// TIA Portal V17 export
// export: Created 2024-08-07T21:43:56.755599Z, ExportSetting WithDefaults, DisplayName Totally Integrated Automation Portal, DisplayVersion V17 Update 7, DisplayName TIA Portal Openness, DisplayVersion V17 Update 7, DisplayName TIA Portal Version Control Interface, DisplayVersion V17, DisplayName SINAMICS Startdrive Advanced, DisplayVersion V17 SP2, DisplayName SINAMICS Startdrive G110M, G120, G120C, G120D, G120P, G115D, DisplayVersion V17 SP2, DisplayName SINAMICS Startdrive G130, G150, S120, S150, SINAMICS MV, S210, DisplayVersion V17 SP2, DisplayName STEP 7 Professional, DisplayVersion V17 Update 7, DisplayName STEP 7 Safety, DisplayVersion V17 Update 6, DisplayName WinCC Advanced / Unified PC, DisplayVersion V17 Update 7
DATA_BLOCK "ScanCompare_DB"   // DB32
VERSION : 0.1
// stored: AutoNumber true, DBAccessibleFromOPCUA true, DBAccessibleFromWebserver true, InstanceOfName ScanCompare, InstanceOfType FB
"ScanCompare"
   // VAR_INPUT
   //    iDMC : String := '';
   //    iStringToCompare : String := '2567208X';
   //    iPosition : Int := 9;
   //    iLength : Int := 8;
   // END_VAR
   // VAR_OUTPUT
   //    comparedString : String := '';
   //    OK : Bool := FALSE;
   // END_VAR
BEGIN
END_DATA_BLOCK
